Omron Sysmac Studio project Motor Control  (Sysmac Studio 1.60.0.64010, StandardProject)

# Controller new_Controller_0: NJ101-1000 version 1.14
Units and slaves: Power Supply : NJ-Px3001; CPU : NJ101-1000
Axis MC_Axis000, settings changed from default: UnitsNumerator=8388608, UnitsDenominator=8388608, MaxJogVelocity=100000
Task PrimaryTask (priority 4, period or condition 2000): Program0

TYPE MyUnion : UNION
    MyWord : WORD;
    MyBits : ARRAY[0..15] OF BOOL;
END_UNION END_TYPE

VAR_GLOBAL
    E001_Controlword : WORD;  (* at ECAT://node#2/Controlword *)
    E001_Target_position : DINT;  (* at ECAT://node#2/Target position *)
    E001_Target_velocity : DINT;  (* at ECAT://node#2/Target velocity *)
    E001_Target_torque : INT;  (* at ECAT://node#2/Target torque *)
    E001_Modes_of_operation : SINT;  (* at ECAT://node#2/Modes of operation *)
    E001_Positive_torque_limit_value : UINT;  (* at ECAT://node#2/Positive torque limit value *)
    E001_Negative_torque_limit_value : UINT;  (* at ECAT://node#2/Negative torque limit value *)
    E001_Statusword : WORD;  (* at ECAT://node#2/Statusword *)
    E001_Position_actual_value : DINT;  (* at ECAT://node#2/Position actual value *)
    G_servolock1 : BOOL;  (* published *)
    G_ResetAll : BOOL;  (* published *)
END_VAR
VAR_GLOBAL CONSTANT
    MC_Axis000 : _sAXIS_REF;  (* at MC://_MC_AX[0] *)
END_VAR

PROGRAM Program0
VAR
    Control_Word : MyUnion;
    E002_Switched_On_Disabled : BOOL;
    Manually_Shutdown : BOOL;
    E002_Fault : BOOL;
    E002_Ready_To_Switch_On : BOOL;
    Manually_Switched_On : BOOL;
    E002_Switched_On : BOOL;
    E002_Operation_Enabled : BOOL;
    ControlWord_Status : MyUnion;
    E002_Not_Ready_To_Switch_On : BOOL;
    E002_Fault_Reaction_Active : BOOL;
    turnon : BOOL;
    RESTE : BOOL;
    test : BOOL;
    skibidi : DINT;
    positionary : ARRAY[0..1] OF DINT;
    train : BOOL;
    indicator : BOOL;
    traingle : LREAL;
    trapezoid : LREAL;
    speedo : ARRAY[0..1] OF DINT;
    acelr : DINT;
    combindis : LREAL;
    automart : BOOL;
    trap : BOOL;
    tringle : BOOL;
    pointer : INT;
    decel : BOOL;
    conversi : BOOL;
    milieter : LREAL;
    timc : TIME;
    disps : LREAL;
    consnp : LREAL;
    timestart : DATE_AND_TIME;
    timeend : DATE_AND_TIME;
    timetaken : DINT;
    ACCEL : DINT;
    fspeed : DINT;
    hawk : BOOL;
    dcalcs : BOOL;
    dval : DINT;
    ACTRI : LREAL;
    DETRI : LREAL;
    trapadd : LREAL;
    trinadd : LREAL;
    square : BOOL;
    squasris : LREAL;
    squart : LREAL;
    dctrl : BOOL;
    b1 : BOOL;
    actrl : BOOL;
    b2 : BOOL;
    intergeal : BOOL;
    period : LREAL;
    grad : ARRAY[0..1] OF LREAL;
    yval : LREAL;
    integ : LREAL;
    totime : LREAL;
    checkspe : LREAL;
    integ2 : LREAL;
    integ3 : LREAL;
    totol : LREAL;
    speedoup : LREAL;
    iteg2 : LREAL;
    iteg3 : LREAL;
    iteg1 : LREAL;
    are1 : LREAL;
    are2 : LREAL;
    are3 : LREAL;
    setdis : LREAL;
    stupid : LREAL;
    count : INT;
    FB_M : MC_Move;
    m : BOOL;
    fspeed_lreal : LREAL;
    a : LREAL;
    accel_lreal : LREAL;
    dv : LREAL;
    dval_lreal : LREAL;
    fb_H : MC_Home;
    H : BOOL;
    SKRULL : BOOL;
    BUTTON : BOOL;
    MOTORATION : MyMove;
    HABA : BOOL;
END_VAR
VAR RETAIN
    pos : LREAL;
    spard : LREAL;
    fast : LREAL;
    slow : LREAL;
END_VAR
VAR
    booger : BOOL;
    MOVE1 : MC_Move;
    ONMOTOR : BOOL;
    START : BOOL;
END_VAR
VAR_EXTERNAL
    E001_Modes_of_operation : SINT;
    E001_Positive_torque_limit_value : UINT;
    E001_Negative_torque_limit_value : UINT;
    G_servolock1 : BOOL;
    G_ResetAll : BOOL;
    E001_Controlword : WORD;
    E001_Statusword : WORD;
    E001_Target_position : DINT;
    E001_Target_velocity : DINT;
    E001_Target_torque : INT;
    E001_Position_actual_value : DINT;
END_VAR
VAR_EXTERNAL CONSTANT
    MC_Axis000 : _sAXIS_REF;
END_VAR
VAR
    _p1 : BOOL;
    _e2 : R_TRIG;
    _e3 : R_TRIG;
    _e4 : R_TRIG;
    _e5 : F_TRIG;
END_VAR

(* Section Section0: ladder, written here as Structured Text *)

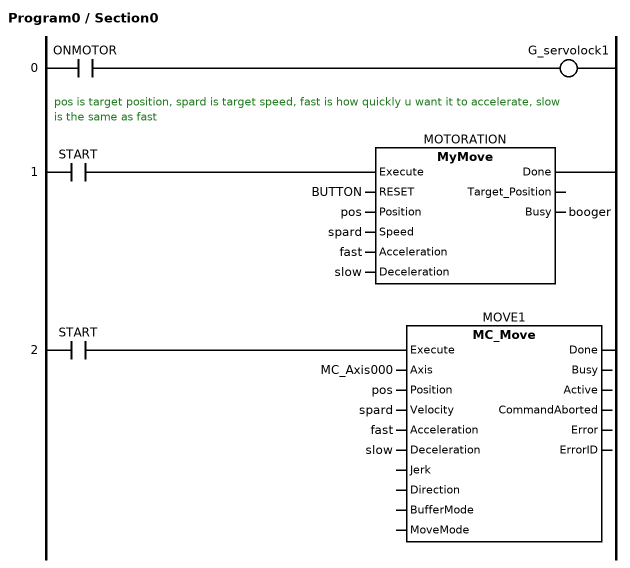
(* Rung 0 *)
G_servolock1 := ONMOTOR;
(* Rung 1: pos is target position, spard is target speed, fast is how quickly u want it to accelerate, slow is the same as fast *)
MOTORATION(Execute := START, RESET := BUTTON, Position := pos, Speed := spard, Acceleration := fast, Deceleration := slow, Busy => booger);
(* Rung 2 *)
MOVE1(Execute := START, Axis := MC_Axis000, Position := pos, Velocity := spard, Acceleration := fast, Deceleration := slow);

(* Section Servolock_wo_MC_Power: ladder, written here as Structured Text *)

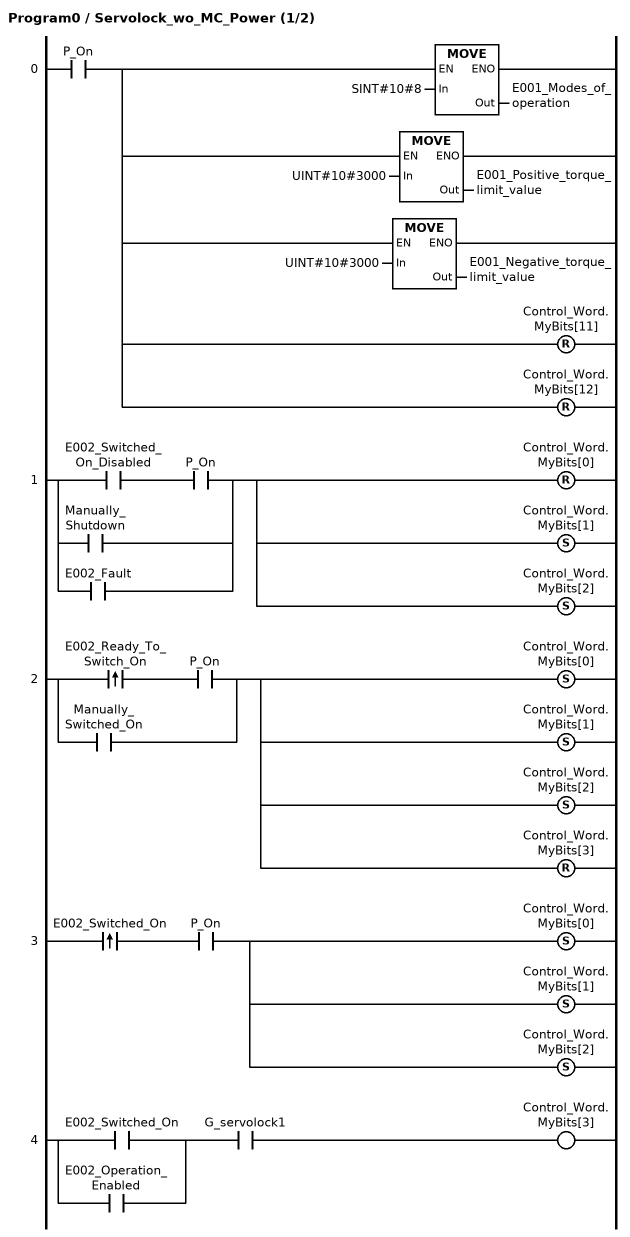
(* Rung 0 *)
IF P_On THEN
    E001_Modes_of_operation := SINT#10#8;
    E001_Positive_torque_limit_value := UINT#10#3000;
    E001_Negative_torque_limit_value := UINT#10#3000;
    Control_Word.MyBits[11] := FALSE;
    Control_Word.MyBits[12] := FALSE;
END_IF;
(* Rung 1 *)
_p1 := (E002_Switched_On_Disabled AND P_On) OR Manually_Shutdown OR E002_Fault;
IF _p1 THEN
    Control_Word.MyBits[0] := FALSE;
    Control_Word.MyBits[1] := TRUE;
    Control_Word.MyBits[2] := TRUE;
END_IF;
(* Rung 2 *)
_e2(CLK := E002_Ready_To_Switch_On);
IF (_e2.Q AND P_On) OR Manually_Switched_On THEN
    Control_Word.MyBits[0] := TRUE;
    Control_Word.MyBits[1] := TRUE;
    Control_Word.MyBits[2] := TRUE;
    Control_Word.MyBits[3] := FALSE;
END_IF;
(* Rung 3 *)
_e3(CLK := E002_Switched_On);
IF _e3.Q AND P_On THEN
    Control_Word.MyBits[0] := TRUE;
    Control_Word.MyBits[1] := TRUE;
    Control_Word.MyBits[2] := TRUE;
END_IF;
(* Rung 4 *)
Control_Word.MyBits[3] := (E002_Switched_On OR E002_Operation_Enabled) AND G_servolock1;

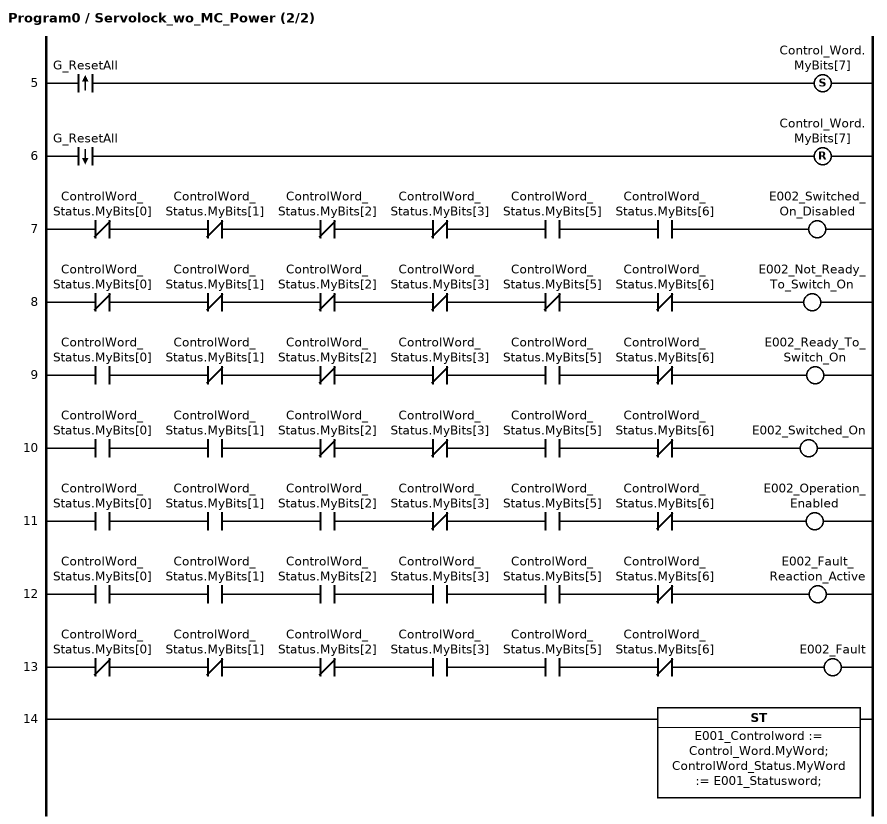
(* Rung 5 *)
_e4(CLK := G_ResetAll);
IF _e4.Q THEN Control_Word.MyBits[7] := TRUE; END_IF;
(* Rung 6 *)
_e5(CLK := G_ResetAll);
IF _e5.Q THEN Control_Word.MyBits[7] := FALSE; END_IF;
(* Rung 7 *)
E002_Switched_On_Disabled := NOT ControlWord_Status.MyBits[0] AND NOT ControlWord_Status.MyBits[1] AND NOT ControlWord_Status.MyBits[2] AND NOT ControlWord_Status.MyBits[3] AND ControlWord_Status.MyBits[5] AND ControlWord_Status.MyBits[6];
(* Rung 8 *)
E002_Not_Ready_To_Switch_On := NOT ControlWord_Status.MyBits[0] AND NOT ControlWord_Status.MyBits[1] AND NOT ControlWord_Status.MyBits[2] AND NOT ControlWord_Status.MyBits[3] AND NOT ControlWord_Status.MyBits[5] AND NOT ControlWord_Status.MyBits[6];
(* Rung 9 *)
E002_Ready_To_Switch_On := ControlWord_Status.MyBits[0] AND NOT ControlWord_Status.MyBits[1] AND NOT ControlWord_Status.MyBits[2] AND NOT ControlWord_Status.MyBits[3] AND ControlWord_Status.MyBits[5] AND NOT ControlWord_Status.MyBits[6];
(* Rung 10 *)
E002_Switched_On := ControlWord_Status.MyBits[0] AND ControlWord_Status.MyBits[1] AND NOT ControlWord_Status.MyBits[2] AND NOT ControlWord_Status.MyBits[3] AND ControlWord_Status.MyBits[5] AND NOT ControlWord_Status.MyBits[6];
(* Rung 11 *)
E002_Operation_Enabled := ControlWord_Status.MyBits[0] AND ControlWord_Status.MyBits[1] AND ControlWord_Status.MyBits[2] AND NOT ControlWord_Status.MyBits[3] AND ControlWord_Status.MyBits[5] AND NOT ControlWord_Status.MyBits[6];
(* Rung 12 *)
E002_Fault_Reaction_Active := ControlWord_Status.MyBits[0] AND ControlWord_Status.MyBits[1] AND ControlWord_Status.MyBits[2] AND ControlWord_Status.MyBits[3] AND ControlWord_Status.MyBits[5] AND NOT ControlWord_Status.MyBits[6];
(* Rung 13 *)
E002_Fault := NOT ControlWord_Status.MyBits[0] AND NOT ControlWord_Status.MyBits[1] AND NOT ControlWord_Status.MyBits[2] AND ControlWord_Status.MyBits[3] AND ControlWord_Status.MyBits[5] AND NOT ControlWord_Status.MyBits[6];
(* Rung 14 *)
E001_Controlword := Control_Word.MyWord;
ControlWord_Status.MyWord := E001_Statusword;
END_PROGRAM

FUNCTION_BLOCK MyMove
VAR
    PLEHLD : BOOL;
    PLCEHLD : BOOL;
    pointer : INT;
    indicator : BOOL;
    automart : BOOL;
    traingle : LREAL;
    trinadd : LREAL;
    trapezoid : LREAL;
    trapadd : LREAL;
    squart : LREAL;
    squasris : LREAL;
    combindis : LREAL;
    positionary : ARRAY[0..1] OF LREAL;
    speedo : ARRAY[0..1] OF LREAL;
    setdis : LREAL;
    fspeed : LREAL;
    ACCEL : LREAL;
    dval : LREAL;
    actrl : BOOL;
    dctrl : BOOL;
    tringle : BOOL;
    trap : BOOL;
    train : BOOL;
    square : BOOL;
    are3 : LREAL;
    decel : BOOL;
    dcalcs : BOOL;
    are1 : LREAL;
    stupid : LREAL;
    are2 : LREAL;
    donezo : BOOL;
    logks : DINT(0..1000000);
    chk : BOOL;
    macaroni : BOOL;
    integ1 : LREAL;
    timering : LINT;
    inter : TIME;
    secondtime : LINT;
    intering : LREAL;
    timber : LREAL;
    indring : LINT;
    integ2 : LREAL;
    hlim : LREAL;
    llim : LREAL;
    binter2 : LREAL;
    BURG : LREAL;
    binter1 : LREAL;
    totalis : LREAL;
    storefinal : LREAL;
    larp : LREAL;
    inval1 : LREAL;
    larg : LREAL;
    inval2 : LREAL;
    inval3 : LREAL;
    tresfina : LREAL;
    ACDCINTEG : LREAL;
    MAIN : BOOL;
    Initialise : BOOL;
    HARDRESET : BOOL;
    Tms : LREAL;
    Tconstant : LREAL;
END_VAR
VAR_INPUT
    Execute : BOOL;
    RESET : BOOL;
    Position : LREAL;
    Speed : LREAL;
    Acceleration : LREAL;
    Deceleration : LREAL;
END_VAR
VAR_OUTPUT
    Done : BOOL;
    Target_Position : DINT;
    Busy : BOOL;
END_VAR
VAR_EXTERNAL
    E001_Target_position : DINT;
    E001_Target_velocity : DINT;
END_VAR
VAR
    _e1 : F_TRIG;
END_VAR
(* ladder, written here as Structured Text *)

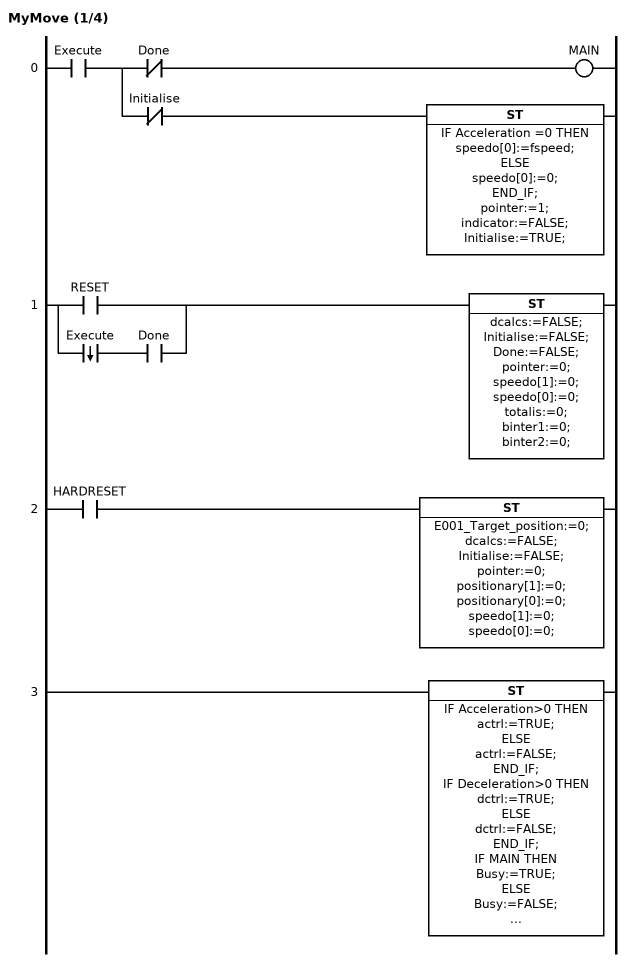
(* Rung 0 *)
MAIN := Execute AND NOT Done;
IF Execute AND NOT Initialise THEN
    IF Acceleration =0 THEN
    	speedo[0]:=fspeed;
    ELSE
    	speedo[0]:=0;
    END_IF;
    pointer:=1;
    indicator:=FALSE;
    
    Initialise:=TRUE;
END_IF;
(* Rung 1 *)
_e1(CLK := Execute);
IF RESET OR (_e1.Q AND Done) THEN
    dcalcs:=FALSE;
    Initialise:=FALSE;
    Done:=FALSE;
    pointer:=0;
    speedo[1]:=0;
    speedo[0]:=0;
    totalis:=0;
    binter1:=0;
    binter2:=0;
END_IF;
(* Rung 2 *)
IF HARDRESET THEN
    E001_Target_position:=0;
    dcalcs:=FALSE;
    Initialise:=FALSE;
    pointer:=0;
    positionary[1]:=0;
    positionary[0]:=0;
    speedo[1]:=0;
    speedo[0]:=0;
END_IF;
(* Rung 3 *)
IF Acceleration>0 THEN
	actrl:=TRUE;
ELSE
	actrl:=FALSE;
END_IF;

IF Deceleration>0 THEN
	dctrl:=TRUE;
ELSE
	dctrl:=FALSE;
END_IF;

IF MAIN THEN
	Busy:=TRUE;
ELSE
	Busy:=FALSE;
END_IF;

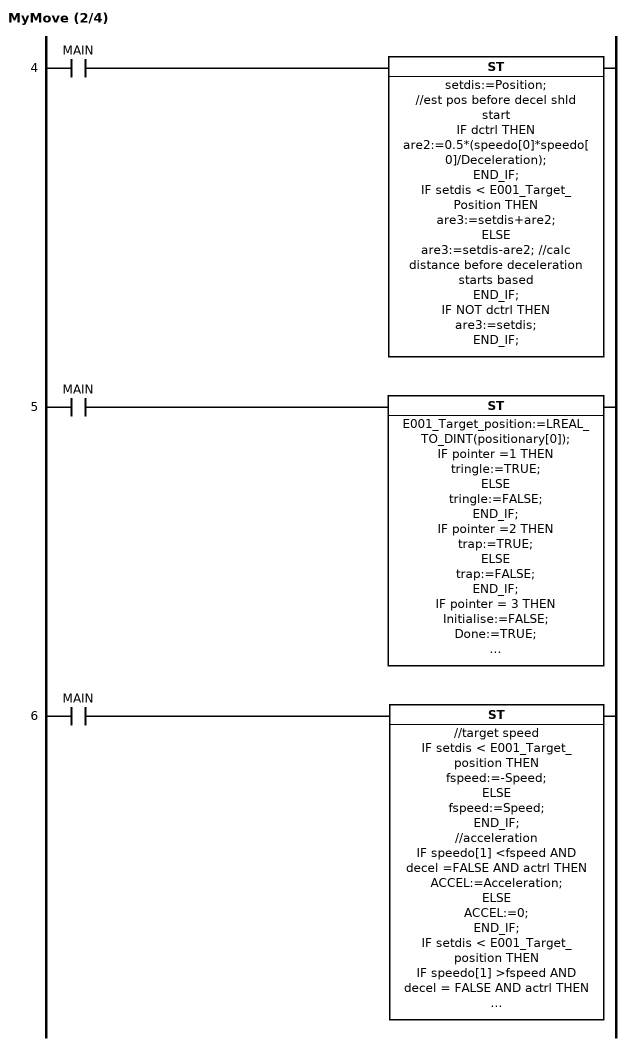
(* Rung 4 *)
IF MAIN THEN
    setdis:=Position;
    
    //est pos before decel shld start
    IF dctrl THEN
    are2:=0.5*(speedo[0]*speedo[0]/Deceleration);
    END_IF;
    IF setdis < E001_Target_Position THEN
    	are3:=setdis+are2;
    ELSE
    	are3:=setdis-are2; //calc distance before deceleration starts based on final d
    END_IF;
    
    IF NOT dctrl THEN
    	are3:=setdis;
    END_IF;
END_IF;
(* Rung 5 *)
IF MAIN THEN
    E001_Target_position:=LREAL_TO_DINT(positionary[0]);
    
    IF pointer =1 THEN
    	tringle:=TRUE;
    ELSE
    	tringle:=FALSE;
    END_IF;
    
    IF pointer =2 THEN
    	trap:=TRUE;
    ELSE
    	trap:=FALSE;
    END_IF;
    
    IF pointer = 3 THEN
    	Initialise:=FALSE;
    	Done:=TRUE;
    END_IF;
    
    IF pointer = 10 THEN
    	square:=TRUE;
    ELSE
    	square:=FALSE;
    END_IF;
    
    
    IF  E001_Target_position >=are3 THEN
    	indicator:=TRUE;
    ELSE
    	indicator:=FALSE;
    END_IF;
    
    IF setdis < E001_Target_position THEN
    	IF  E001_Target_position <=are3 THEN
    	indicator:=TRUE;
    ELSE
    	indicator:=FALSE;
    END_IF;
    END_IF;
    
    
    ArySHL(positionary[0], 2, 1);
    
    positionary[0]:=positionary[1]+(speedo[0]/Tconstant);
    
    ArySHL(speedo[0], 2, 1);
END_IF;
(* Rung 6 *)
IF MAIN THEN
    //target speed
    	
    	IF setdis < E001_Target_position THEN
    		fspeed:=-Speed;
    	ELSE
    		fspeed:=Speed;
    	END_IF;
    
    //acceleration
    IF speedo[1] <fspeed AND decel =FALSE AND actrl THEN
    	ACCEL:=Acceleration;
    ELSE
    	ACCEL:=0;
    END_IF;
    IF setdis < E001_Target_position THEN
    	IF speedo[1] >fspeed AND decel = FALSE AND actrl THEN
    		ACCEL:=-Acceleration;
    	ELSE
    		ACCEL:=0;
    	END_IF;
    END_IF;
    
    //change deceleration
    IF dcalcs AND setdis < E001_Target_position THEN
    	dval:=-Deceleration;
    ELSIF dcalcs THEN
    	dval:=Deceleration;
    ELSE
    	dval:=0;
    END_IF;
    
    hlim:= MAX(ACCEL,dval);
    llim:=MIN(-ACCEL,-dval);
    
    speedo[0] := LIMIT(llim, speedo[0], hlim);
    
    speedo[0]:=(speedo[1]+(ACCEL/Tconstant)-(dval/Tconstant));
END_IF;

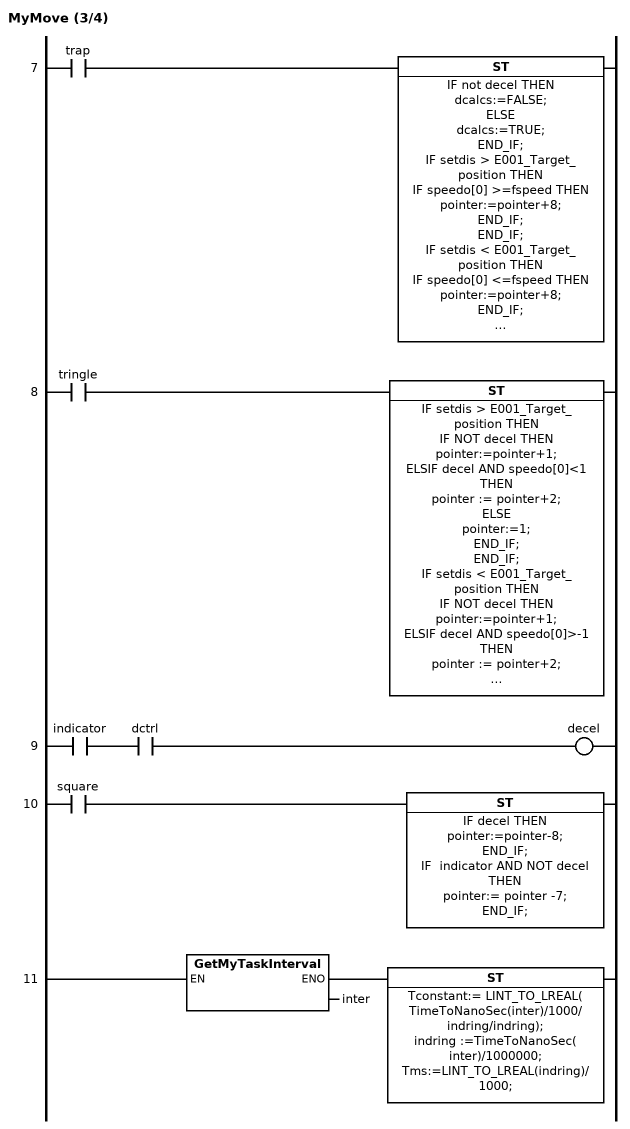
(* Rung 7 *)
IF trap THEN
    IF not decel THEN
    	dcalcs:=FALSE;
    ELSE
    	dcalcs:=TRUE;
    END_IF;
    
    IF setdis > E001_Target_position THEN
    	IF speedo[0] >=fspeed THEN
    		pointer:=pointer+8;
    	END_IF;
    END_IF;
    
    IF setdis < E001_Target_position THEN
    	IF speedo[0] <=fspeed THEN
    		pointer:=pointer+8;
    	END_IF;
    END_IF;
    
    IF setdis > E001_Target_position THEN
    	IF decel=1 AND speedo[0] <1 THEN
    		pointer:=pointer-1;
    	END_IF;
    END_IF;
    
    IF setdis<E001_Target_position THEN
    	IF decel =1 AND speedo[0]>-1 THEN
    		pointer:=pointer-1;
    	END_IF;
    END_IF;
END_IF;
(* Rung 8 *)
IF tringle THEN
    IF setdis > E001_Target_position THEN
    	IF NOT decel THEN
    		pointer:=pointer+1;
    	ELSIF decel AND speedo[0]<1 THEN
    		pointer := pointer+2;
    	ELSE
    		pointer:=1;
    	END_IF;
    END_IF;
    
    IF setdis < E001_Target_position THEN
    	IF NOT decel THEN
    		pointer:=pointer+1;
    	ELSIF decel AND speedo[0]>-1 THEN
    		pointer := pointer+2;
    	ELSE
    		pointer:=1;
    	END_IF;
    END_IF;
    
    IF actrl = FALSE and not decel THEN
    	pointer:=pointer+8;
    END_IF;
END_IF;
(* Rung 9 *)
decel := indicator AND dctrl;
(* Rung 10 *)
IF square THEN
    IF decel THEN
    	pointer:=pointer-8;
    END_IF;
    
    IF  indicator AND NOT decel THEN
    	pointer:= pointer -7;
    END_IF;
END_IF;
(* Rung 11 *)
inter := GetMyTaskInterval();
Tconstant:= LINT_TO_LREAL(TimeToNanoSec(inter)/1000/indring/indring);
indring :=TimeToNanoSec(inter)/1000000;
Tms:=LINT_TO_LREAL(indring)/1000;

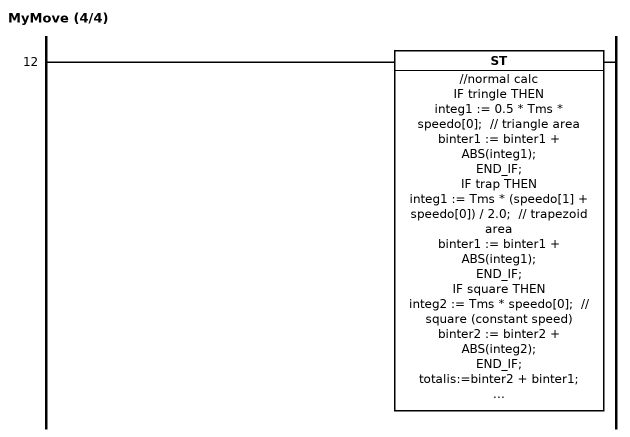
(* Rung 12 *)
//normal calc
IF tringle THEN
    integ1 := 0.5 * Tms * speedo[0];  // triangle area
    binter1 := binter1 + ABS(integ1);
END_IF;

IF trap THEN
    integ1 := Tms * (speedo[1] + speedo[0]) / 2.0;  // trapezoid area
    binter1 := binter1 + ABS(integ1);
END_IF;

IF square THEN
    integ2 := Tms * speedo[0];  // square (constant speed)
    binter2 := binter2 + ABS(integ2);
END_IF;

totalis:=binter2 + binter1;

//integration
ACDCINTEG:= ACDCINTEG+Tms*speedo[1];
END_FUNCTION_BLOCK